// TIA Portal project "LAST TEST PMW" (V16)

(* hardware
DEVICE "S7-1200 station_1"  S7-1200 Station
   slot 0: "Rack_0"  S7-1200 Rack  Rack  V1.0
   slot 1: "PLC_1"  CPU 1214C DC/DC/DC  6ES7 214-1AG40-0XB0  V4.2
   slot 2: "AI 4x13BIT/AQ 2x14BIT_1"  6ES7 234-4HE32-0XB0  V2.1
*)

// ===== PLC "PLC_1"  CPU 1214C DC/DC/DC =====

VAR_GLOBAL   // PLC tag table "Default tag table"
   "SENSOR TANK 1" AT %IW64 : Int;
   "PUMP 1" AT %QW98 : Int;
   "PV 1 DATA" AT %MD2 : Real;
   "SETPOINT" AT %MW0 : Int;
   "PV 2 DATA" AT %MD4 : DWord;
   "DATA PV TANK 1 C" AT %MD6 : Real;
   "SENSOR TANK 2" AT %IW66 : Int;
   "DATA MV PID 2 TO TCP" AT %MD8 : DWord;
   "PV TANK 2 TO WECON" AT %MW12 : Int;
   "MV PID 1 TO WECON" AT %MW14 : Int;
   "MV PID 2 TO WECON" AT %MW16 : Int;
   "PV TANK 1 TO WECON" AT %MW18 : Int;
   "Tag_2" AT %Q0.0 : Bool;
   "Tag_1" AT %Q0.1 : Bool;
   "Tag_3" AT %Q0.2 : Bool;
   "Tag_4" AT %M30.0 : Bool;
   "Tag_5" AT %M32.0 : Bool;
   "Tag_6" AT %M34.0 : Bool;
END_VAR

DATA_BLOCK "DATA_PID"   // DB2
{ S7_Optimized_Access := 'TRUE' }
VERSION : 0.1
   VAR
      "SP TANK 2" : Real;
      "PV TANK 1" : Real;
      "PV TANK 2" : Real;
      "MV PID 1" : Real;
      "MV PID 2" : Real;
      "PV TANK 1 C" : Real;
      "MV PID 2 OUTP" : Real;
   END_VAR
BEGIN
END_DATA_BLOCK

DATA_BLOCK "DATA TCP"   // DB4
{ S7_Optimized_Access := 'FALSE' }
VERSION : 0.1
   VAR
      DATA : Array[0..4] of Int;
   END_VAR
BEGIN
END_DATA_BLOCK

DATA_BLOCK "MB config"   // DB6
{ S7_Optimized_Access := 'FALSE' }
VERSION : 0.1
   VAR
      CONNECT : TCON_IP_v4;
   END_VAR
BEGIN
   CONNECT.InterfaceId := 64;
   CONNECT.ID := 1;
   CONNECT.ConnectionType := 11;
   CONNECT.RemoteAddress.ADDR[1] := 192;
   CONNECT.RemoteAddress.ADDR[2] := 168;
   CONNECT.RemoteAddress.ADDR[3] := 0;
   CONNECT.RemoteAddress.ADDR[4] := 100;
   CONNECT.LocalPort := 502;
END_DATA_BLOCK

// folder: System blocks/Program resources

DATA_BLOCK "IEC_Timer_0_DB"   // DB7
{ S7_Optimized_Access := 'TRUE' }
AUTHOR : Simatic
FAMILY : IEC
NAME : IEC_TMR
VERSION : 1.0
// stored: InstanceOfName IEC_TIMER
"IEC_TIMER"
BEGIN
END_DATA_BLOCK

DATA_BLOCK "IEC_Timer_0_DB_1"   // DB8
{ S7_Optimized_Access := 'TRUE' }
AUTHOR : Simatic
FAMILY : IEC
NAME : IEC_TMR
VERSION : 1.0
// stored: InstanceOfName IEC_TIMER
"IEC_TIMER"
BEGIN
END_DATA_BLOCK

DATA_BLOCK "IEC_Timer_0_DB_2"   // DB9
{ S7_Optimized_Access := 'TRUE' }
AUTHOR : Simatic
FAMILY : IEC
NAME : IEC_TMR
VERSION : 1.0
// stored: InstanceOfName IEC_TIMER
"IEC_TIMER"
BEGIN
END_DATA_BLOCK

// folder: (top level)

FUNCTION "Sceal" : Void   // FC1, LAD
{ S7_Optimized_Access := 'TRUE' }
VERSION : 0.1
BEGIN

REGION Network 1: SENSOR 1
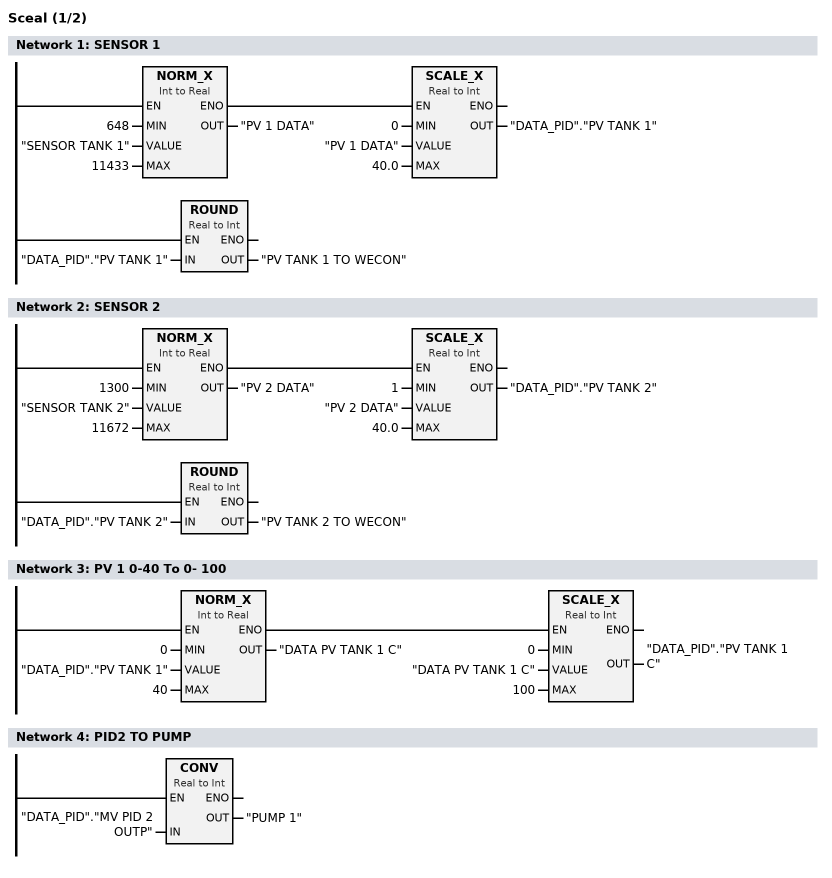
   RUNG wire#powerrail
      { S7_Templates := "[SrcType := Int, DestType := Real]" } Normalize(min := 648, value := "SENSOR TANK 1", max := 11433, out => "PV 1 DATA")
      { S7_Templates := "[SrcType := Real, DestType := Int]" } Scale(min := 0, value := "PV 1 DATA", max := 40.0, out => "DATA_PID"."PV TANK 1")
   END_RUNG
   RUNG wire#powerrail
      { S7_Templates := "[SrcType := Real, DestType := Int]" } Round(in := "DATA_PID"."PV TANK 1", out => "PV TANK 1 TO WECON")
   END_RUNG
   // the same network as SCL:
   "PV 1 DATA" := NORM_X(MIN := 648, VALUE := "SENSOR TANK 1", MAX := 11433);
   "DATA_PID"."PV TANK 1" := SCALE_X(MIN := 0, VALUE := "PV 1 DATA", MAX := 40.0);
   "PV TANK 1 TO WECON" := ROUND("DATA_PID"."PV TANK 1");
END_REGION

REGION Network 2: SENSOR 2
   RUNG wire#powerrail
      { S7_Templates := "[SrcType := Int, DestType := Real]" } Normalize(min := 1300, value := "SENSOR TANK 2", max := 11672, out => "PV 2 DATA")
      { S7_Templates := "[SrcType := Real, DestType := Int]" } Scale(min := 1, value := "PV 2 DATA", max := 40.0, out => "DATA_PID"."PV TANK 2")
   END_RUNG
   RUNG wire#powerrail
      { S7_Templates := "[SrcType := Real, DestType := Int]" } Round(in := "DATA_PID"."PV TANK 2", out => "PV TANK 2 TO WECON")
   END_RUNG
   // the same network as SCL:
   "PV 2 DATA" := NORM_X(MIN := 1300, VALUE := "SENSOR TANK 2", MAX := 11672);
   "DATA_PID"."PV TANK 2" := SCALE_X(MIN := 1, VALUE := "PV 2 DATA", MAX := 40.0);
   "PV TANK 2 TO WECON" := ROUND("DATA_PID"."PV TANK 2");
END_REGION

REGION Network 3: PV 1 0-40 To 0- 100
   RUNG wire#powerrail
      { S7_Templates := "[SrcType := Int, DestType := Real]" } Normalize(min := 0, value := "DATA_PID"."PV TANK 1", max := 40, out => "DATA PV TANK 1 C")
      { S7_Templates := "[SrcType := Real, DestType := Int]" } Scale(min := 0, value := "DATA PV TANK 1 C", max := 100, out => "DATA_PID"."PV TANK 1 C")
   END_RUNG
   // the same network as SCL:
   "DATA PV TANK 1 C" := NORM_X(MIN := 0, VALUE := "DATA_PID"."PV TANK 1", MAX := 40);
   "DATA_PID"."PV TANK 1 C" := SCALE_X(MIN := 0, VALUE := "DATA PV TANK 1 C", MAX := 100);
END_REGION

REGION Network 4: PID2 TO PUMP
   RUNG wire#powerrail
      { S7_Templates := "[SrcType := Real, DestType := Int]" } Convert(in := "DATA_PID"."MV PID 2 OUTP", out => "PUMP 1")
   END_RUNG
   // the same network as SCL:
   "PUMP 1" := REAL_TO_INT("DATA_PID"."MV PID 2 OUTP");
END_REGION

REGION Network 5: TO TCP
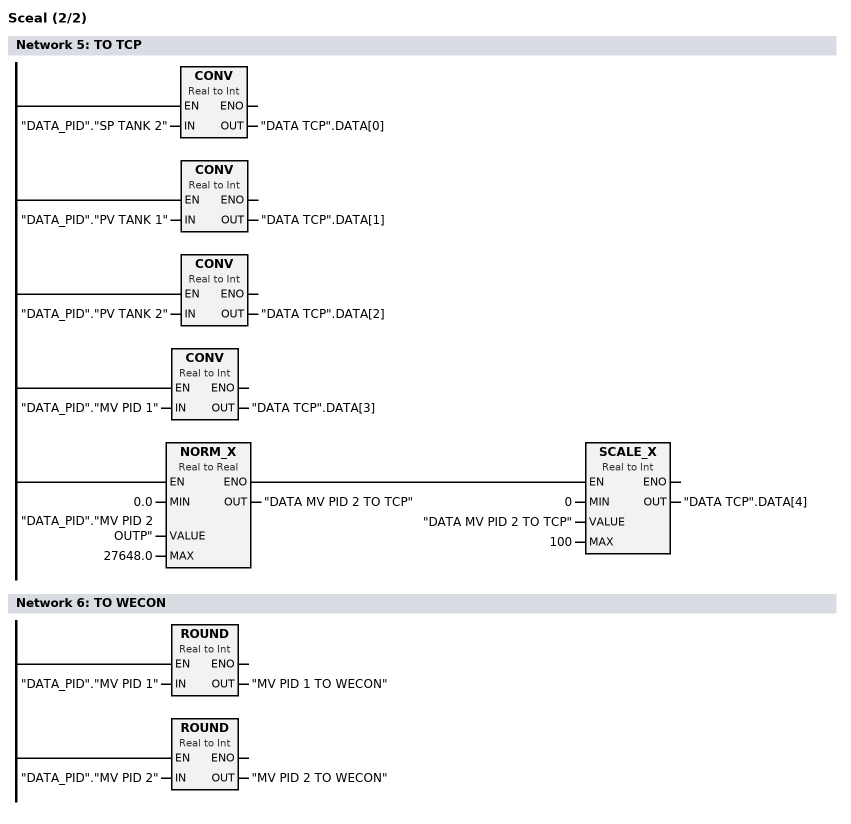
   RUNG wire#powerrail
      { S7_Templates := "[SrcType := Real, DestType := Int]" } Convert(in := "DATA_PID"."SP TANK 2", out => "DATA TCP".DATA[0])
   END_RUNG
   RUNG wire#powerrail
      { S7_Templates := "[SrcType := Real, DestType := Int]" } Convert(in := "DATA_PID"."PV TANK 1", out => "DATA TCP".DATA[1])
   END_RUNG
   RUNG wire#powerrail
      { S7_Templates := "[SrcType := Real, DestType := Int]" } Convert(in := "DATA_PID"."PV TANK 2", out => "DATA TCP".DATA[2])
   END_RUNG
   RUNG wire#powerrail
      { S7_Templates := "[SrcType := Real, DestType := Int]" } Convert(in := "DATA_PID"."MV PID 1", out => "DATA TCP".DATA[3])
   END_RUNG
   RUNG wire#powerrail
      { S7_Templates := "[SrcType := Real, DestType := Real]" } Normalize(min := 0.0, value := "DATA_PID"."MV PID 2 OUTP", max := 27648.0, out => "DATA MV PID 2 TO TCP")
      { S7_Templates := "[SrcType := Real, DestType := Int]" } Scale(min := 0, value := "DATA MV PID 2 TO TCP", max := 100, out => "DATA TCP".DATA[4])
   END_RUNG
   // the same network as SCL:
   "DATA TCP".DATA[0] := REAL_TO_INT("DATA_PID"."SP TANK 2");
   "DATA TCP".DATA[1] := REAL_TO_INT("DATA_PID"."PV TANK 1");
   "DATA TCP".DATA[2] := REAL_TO_INT("DATA_PID"."PV TANK 2");
   "DATA TCP".DATA[3] := REAL_TO_INT("DATA_PID"."MV PID 1");
   "DATA MV PID 2 TO TCP" := NORM_X(MIN := 0.0, VALUE := "DATA_PID"."MV PID 2 OUTP", MAX := 27648.0);
   "DATA TCP".DATA[4] := SCALE_X(MIN := 0, VALUE := "DATA MV PID 2 TO TCP", MAX := 100);
END_REGION

REGION Network 6: TO WECON
   RUNG wire#powerrail
      { S7_Templates := "[SrcType := Real, DestType := Int]" } Round(in := "DATA_PID"."MV PID 1", out => "MV PID 1 TO WECON")
   END_RUNG
   RUNG wire#powerrail
      { S7_Templates := "[SrcType := Real, DestType := Int]" } Round(in := "DATA_PID"."MV PID 2", out => "MV PID 2 TO WECON")
   END_RUNG
   // the same network as SCL:
   "MV PID 1 TO WECON" := ROUND("DATA_PID"."MV PID 1");
   "MV PID 2 TO WECON" := ROUND("DATA_PID"."MV PID 2");
END_REGION
END_FUNCTION

ORGANIZATION_BLOCK "Main"   // OB1, LAD, ProgramCycle
TITLE = "Main Program Sweep (Cycle)"
{ S7_Optimized_Access := 'TRUE' }
VERSION : 0.1
   VAR_INPUT
      Initial_Call : Bool;   // Initial call of this OB
      Remanence : Bool;   // =True, if remanent data are available
   END_VAR
BEGIN

REGION Network 1
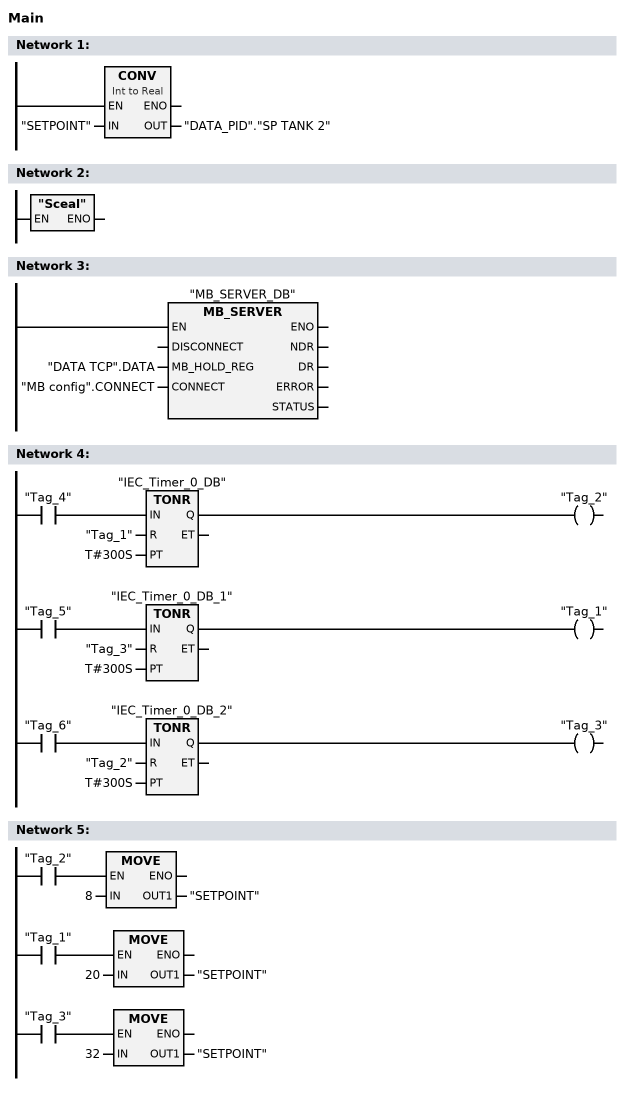
   RUNG wire#powerrail
      { S7_Templates := "[SrcType := Int, DestType := Real]" } Convert(in := "SETPOINT", out => "DATA_PID"."SP TANK 2")
   END_RUNG
   // the same network as SCL:
   "DATA_PID"."SP TANK 2" := INT_TO_REAL("SETPOINT");
END_REGION

REGION Network 2
   RUNG wire#powerrail
      "Sceal"()
   END_RUNG
   // the same network as SCL:
   "Sceal"();
END_REGION

REGION Network 3
   "MB_SERVER_DB"(MB_HOLD_REG := "DATA TCP".DATA, CONNECT := "MB config".CONNECT);   // MB_SERVER
END_REGION

REGION Network 4
   "IEC_Timer_0_DB".TONR(IN := "Tag_4", R := "Tag_1", PT := T#300S);
   "Tag_2" := "IEC_Timer_0_DB".Q;
   "IEC_Timer_0_DB_1".TONR(IN := "Tag_5", R := "Tag_3", PT := T#300S);
   "Tag_1" := "IEC_Timer_0_DB_1".Q;
   "IEC_Timer_0_DB_2".TONR(IN := "Tag_6", R := "Tag_2", PT := T#300S);
   "Tag_3" := "IEC_Timer_0_DB_2".Q;
END_REGION

REGION Network 5
   RUNG wire#powerrail
      Contact( "Tag_2" )
      Move(in := 8, out1 => "SETPOINT")
   END_RUNG
   RUNG wire#powerrail
      Contact( "Tag_1" )
      Move(in := 20, out1 => "SETPOINT")
   END_RUNG
   RUNG wire#powerrail
      Contact( "Tag_3" )
      Move(in := 32, out1 => "SETPOINT")
   END_RUNG
   // the same network as SCL:
   IF "Tag_2" THEN "SETPOINT" := 8; END_IF;
   IF "Tag_1" THEN "SETPOINT" := 20; END_IF;
   IF "Tag_3" THEN "SETPOINT" := 32; END_IF;
END_REGION
END_ORGANIZATION_BLOCK

ORGANIZATION_BLOCK "Cyclic interrupt"   // OB30, LAD, CyclicInterrupt
{ S7_Optimized_Access := 'TRUE' }
VERSION : 0.1
   VAR_INPUT
      Initial_Call : Bool;   // Initial call of this OB
      Event_Count : Int;   // Events discarded
   END_VAR
BEGIN

REGION Network 1
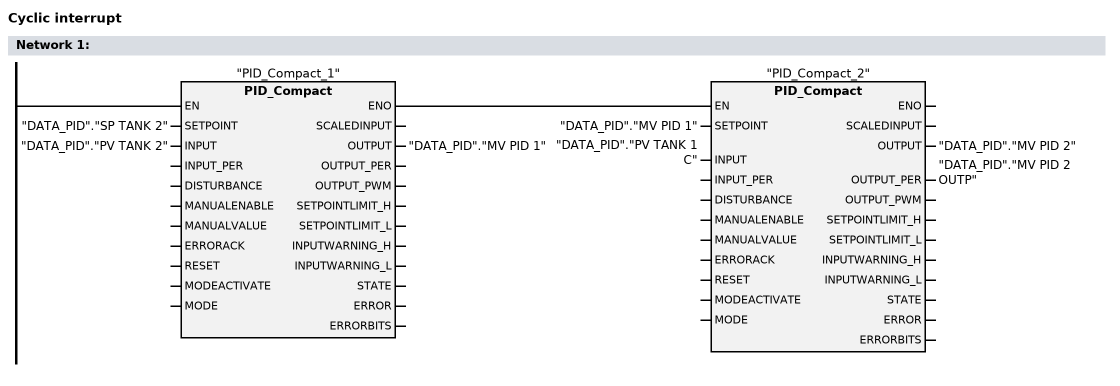
   // ENO of a box is taken as its EN; it also drops when the box reports an error
   "PID_Compact_1"(Setpoint := "DATA_PID"."SP TANK 2",   // PID_Compact
                   Input := "DATA_PID"."PV TANK 2",
                   Output => "DATA_PID"."MV PID 1");
   "PID_Compact_2"(Setpoint := "DATA_PID"."MV PID 1",   // PID_Compact
                   Input := "DATA_PID"."PV TANK 1 C",
                   Output => "DATA_PID"."MV PID 2",
                   Output_PER => "DATA_PID"."MV PID 2 OUTP");
END_REGION
END_ORGANIZATION_BLOCK